FUNCTION_BLOCK Test_F_DateAsString_ReturnsDateString EXTENDS TUnitTestBase
VAR
    TimeStruct : TIMESTRUCT := (wDay := 23, wMonth := 12, wYear := 1945);
END_VAR

Assertion.AssertEquals_STRING(
    Expected := '23/12/1945',
    Actual   := F_DateAsString(TimeStruct),
    VariableName  := 'F_DateAsString(TimeStruct)');


TestFinished();

END_FUNCTION_BLOCK

(* stored: Version 1.1.0.1, ProductVersion 3.1.4024.4
   POU Test_F_DateAsString_ReturnsDateString: Id {dbb0c8d6-f694-0d2d-11c0-291b7b634d6f}, SpecialFunc None *)
